FUNCTION F_CheckInRange : bool
VAR_INPUT
	lrHighLimit	: LREAL;
	lrLowLimit	: LREAL;
	lrValue		: LREAL;
END_VAR
VAR
END_VAR

IF lrLowLimit<=  lrValue AND lrValue <= lrHighLimit THEN
	F_CheckInRange := TRUE;
ELSE 
	F_CheckInRange := FALSE;
END_IF

END_FUNCTION

(* stored: Version 1.1.0.1, ProductVersion 3.1.4024.12
   POU F_CheckInRange: Id {19204482-20e5-4bfe-aea2-8da44390ea24}, SpecialFunc None *)
